// TIA Portal project "PRUEBAS" (V15)

(* hardware
DEVICE "S7-1200 station_1"  S7-1200 Station
   slot 0: "Rack_0"  S7-1200 Rack  Rack  V1.0
   slot 1: "PLC_1"  CPU 1215C AC/DC/Rly  6ES7 215-1BG40-0XB0  V4.2
*)

// ===== PLC "PLC_1"  CPU 1215C AC/DC/Rly =====

VAR_GLOBAL   // PLC tag table "Tabla de variables estándar"
   "Entrada" AT %I0.1 : Bool;
   "Velocidad" AT %MD100 : Real;
   "H" AT %MD800 : Real;
   "Salida" AT %QW64 : Int;
   "Motor_on" AT %M400.0 : Bool;
   "Etapa_1" AT %M200.1 : Bool;
   "Etapa_3" AT %M200.3 : Bool;
   "Etapa_4" AT %M200.4 : Bool;
   "Etapa_5" AT %M200.5 : Bool;
   "pp" AT %M600.0 : Bool;
   "selector" AT %M600.1 : Bool;
   "P" AT %MD750 : Real;
   "SH" AT %MD650 : Real;
END_VAR

ORGANIZATION_BLOCK "Main"   // OB1, LAD, ProgramCycle
TITLE = "Main Program Sweep (Cycle)"
{ S7_Optimized_Access := 'TRUE' }
VERSION : 0.1
   VAR_INPUT
      Initial_Call : Bool;   // Initial call of this OB
      Remanence : Bool;   // =True, if remanent data are available
   END_VAR
BEGIN

REGION Network 1
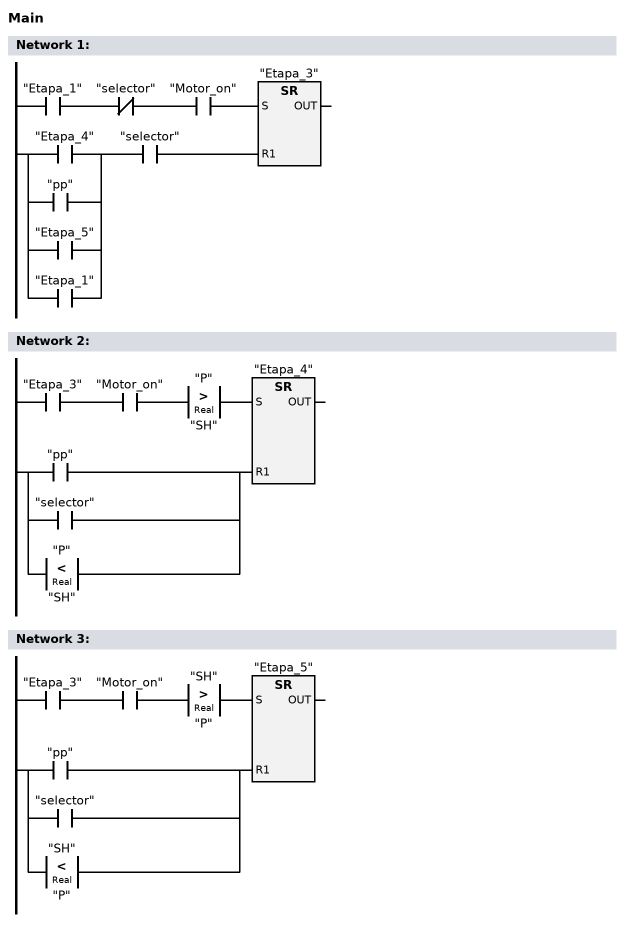
   RUNG wire#powerrail
      Contact( "Etapa_1" )
      I_Contact( "selector" )
      Contact( "Motor_on" )
      S_SR(operand := "Etapa_3", r1 := wire#w2)
   END_RUNG
   RUNG wire#powerrail
      Contact( "Etapa_4" )
      wire#w1
      Contact( "selector" )
   END_RUNG wire#w2
   RUNG wire#powerrail
      Contact( "pp" )
   END_RUNG wire#w1
   RUNG wire#powerrail
      Contact( "Etapa_5" )
   END_RUNG wire#w1
   RUNG wire#powerrail
      Contact( "Etapa_1" )
   END_RUNG wire#w1
   // the same network as SCL:
   IF "Etapa_1" AND NOT "selector" AND "Motor_on" THEN
       "Etapa_3" := TRUE;   // SR flip-flop
   END_IF;
   IF ("Etapa_4" OR "pp" OR "Etapa_5" OR "Etapa_1") AND "selector" THEN "Etapa_3" := FALSE; END_IF;
END_REGION

REGION Network 2
   RUNG wire#powerrail
      Contact( "Etapa_3" )
      Contact( "Motor_on" )
      { S7_Templates := "SrcType := Real" } GT_Contact(in1 := "P", in2 := "SH")
      S_SR(operand := "Etapa_4", r1 := wire#w1)
   END_RUNG
   RUNG wire#powerrail
      Contact( "pp" )
   END_RUNG wire#w1
   RUNG wire#powerrail
      Contact( "selector" )
   END_RUNG wire#w1
   RUNG wire#powerrail
      { S7_Templates := "SrcType := Real" } LT_Contact(in1 := "P", in2 := "SH")
   END_RUNG wire#w1
   // the same network as SCL:
   IF "Etapa_3" AND "Motor_on" AND ("P" > "SH") THEN
       "Etapa_4" := TRUE;   // SR flip-flop
   END_IF;
   IF "pp" OR "selector" OR ("P" < "SH") THEN "Etapa_4" := FALSE; END_IF;
END_REGION

REGION Network 3
   RUNG wire#powerrail
      Contact( "Etapa_3" )
      Contact( "Motor_on" )
      { S7_Templates := "SrcType := Real" } GT_Contact(in1 := "SH", in2 := "P")
      S_SR(operand := "Etapa_5", r1 := wire#w1)
   END_RUNG
   RUNG wire#powerrail
      Contact( "pp" )
   END_RUNG wire#w1
   RUNG wire#powerrail
      Contact( "selector" )
   END_RUNG wire#w1
   RUNG wire#powerrail
      { S7_Templates := "SrcType := Real" } LT_Contact(in1 := "SH", in2 := "P")
   END_RUNG wire#w1
   // the same network as SCL:
   IF "Etapa_3" AND "Motor_on" AND ("SH" > "P") THEN
       "Etapa_5" := TRUE;   // SR flip-flop
   END_IF;
   IF "pp" OR "selector" OR ("SH" < "P") THEN "Etapa_5" := FALSE; END_IF;
END_REGION
END_ORGANIZATION_BLOCK